PROGRAM Internal_Mapping
VAR
	CKKALARMRESET: BOOL;
	CKKBUZZERRESET: BOOL;
	
END_VAR

//ARwDO[eY11002_GeneralBuzzerTone01].00:=bBuzzerOutput; // Need to mapping with pyshical Output Buzzer Tone 1

//bEventRstPBPhysicalInput:=ARbDI[eX10000_Stn01UltrasonicGeneratorMcb_Trip] OR CKKALARMRESET OR bHMI_AlarmRstPB;  // Need to mapping with physical Input Alarm Reset PB
//bBuzzerRstPBPhysicalInput:=ARbDI[eX10001_GeneralBuzzerPb_Reset] OR CKKBUZZERRESET OR bHMI_BuzzerRstPB; // Need to mapping with physical Input Buzzer Reset PB


// Clangsonic Ultrasonic Mapping
//ARdsClangsonicGenerator[1].iGenModbusUnitID		:= 1;
//ARdsClangsonicGenerator[2].iGenModbusUnitID		:= 2;
//ARdsClangsonicGenerator[3].iGenModbusUnitID		:= 3;

//ARdsClangsonicGenerator[1].iModbusRS485ChannelID	:= 1;
//ARdsClangsonicGenerator[2].iModbusRS485ChannelID	:= 1;
//ARdsClangsonicGenerator[3].iModbusRS485ChannelID	:= 1;


// Misshook Sensor

	ARbMAP_ArmMisshookSensorA[1]	:= ARbDI[eX11004_Arm01SensorA_Misshook];
	ARbMAP_ArmMisshookSensorB[1]	:= ARbDI[eX11005_Arm01SensorB_Misshook];
	

//  Last index basket at loading ( Basket LD arm pick )

	bMAP_LdConfirmBasketPickAvailibility   := AR2sDSCv_LdConfirmBasketInfo[1,3].bAvailibility;

END_PROGRAM

(* stored: Version 1.1.0.1, ProductVersion 3.1.4024.12
   POU Internal_Mapping: Id {a6b33a70-f6c9-4aca-a064-f4bef62ee907}, SpecialFunc None *)
